// TIA Portal V19 export
TYPE "TAx_Config"
// stored: Access Published
   STRUCT
      Simulation : Bool;
      PowerOffDelay : Time := T#10s;   // Power off delay with no cmd
      PowerStartMode : Int := 1;   // 0=Non position controlled mode; 1=Position controlled mode
      PowerStopMode : Int := 2;   // 0=Emergency Stop; 1=Quick Stop with OFF3, 2=Stop with max dynamics, 3=Coast Down
   END_STRUCT;
END_TYPE
